ABB RobotStudio station: 20204 CCSU ROS EGM.rspag

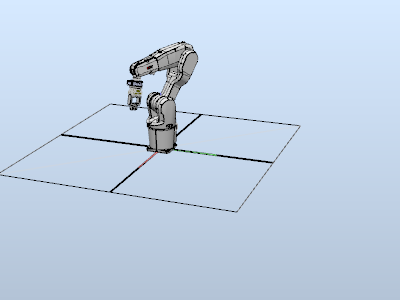
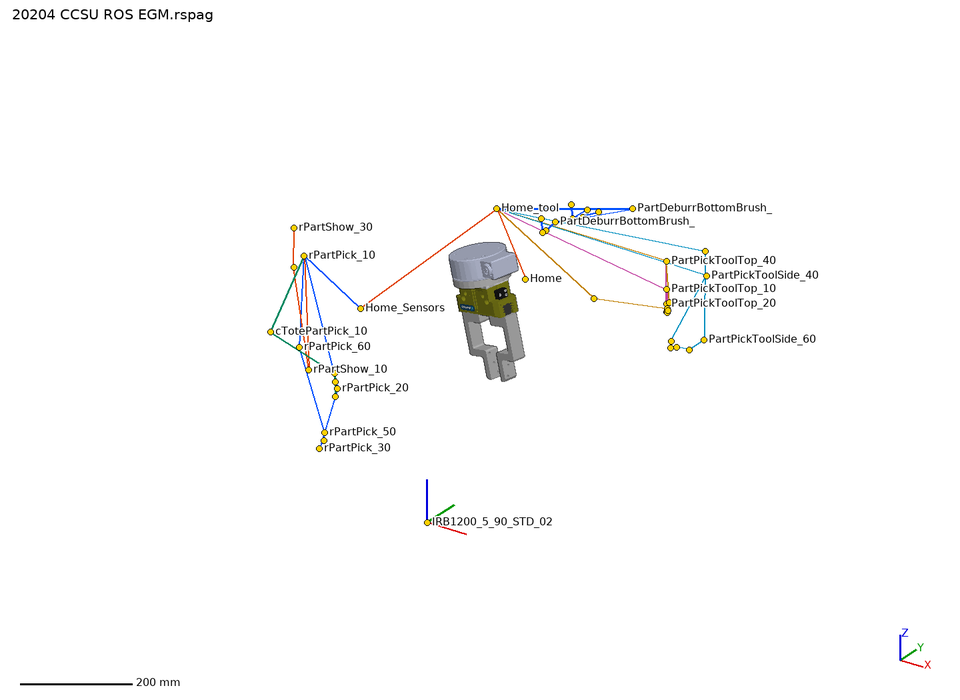
[picture v1: parts stored in the station drawn from their meshes, with robot base, taught points and paths (robot models come from the ABB library and are not in the file)]
--- station ---
Station 20204 CCSU RS (saved by RobotStudio 22.3.10098.0)
Controller 1200-800743_OfflineStation
  mechanical unit ROB_1: IRB1200_5_90_STD_02, 6 joints, base frame (0, 0, 0) mm
Layout (positions relative to the parent item):
  - IRB1200_5_90_STD_02 [mechanism, from %ABB.RobotStudio.Models.IRB1200%\IRB1200_5_90_STD_03.rslib] at (0, 0, 0) mm; joint values [-0.6243, -0.5477, 0.7485, -3.0114, -1.1483, -1.9775] (rad or m)
  - GRIPPER ONLY [part] at (196.51, -129.61, 653.41) mm, rotated rx -178.16 ry -14.43 rz -15 deg, size 125.6 x 50 x 198.4 mm
  - GRIPPER FORCE SENSOR [part] at (196.51, -129.61, 653.41) mm, rotated rx -178.16 ry -14.43 rz -15 deg, size 142.7 x 104 x 238.4 mm
Attachment: GRIPPER ONLY is attached to IRB1200_5_90_STD_02 / Link6
Attachment: GRIPPER FORCE SENSOR is attached to IRB1200_5_90_STD_02 / Link6
Targets, tools, work objects and paths stored in the station and not in the controller backup, written as RAPID:
! task T_ROB1
MODULE FORCENewProgram
  CONST robtarget GoHome:=[[-163.21,-220.75,679.83],[0.000017864,-0.460993,0.887404,0.000003505],[-2,0,1,0],[9E+09,9E+09,9E+09,9E+09,9E+09,9E+09]];
  PROC rGoHome()
    MoveJ GoHome,v500,z50,tool0;
  ENDPROC
ENDMODULE


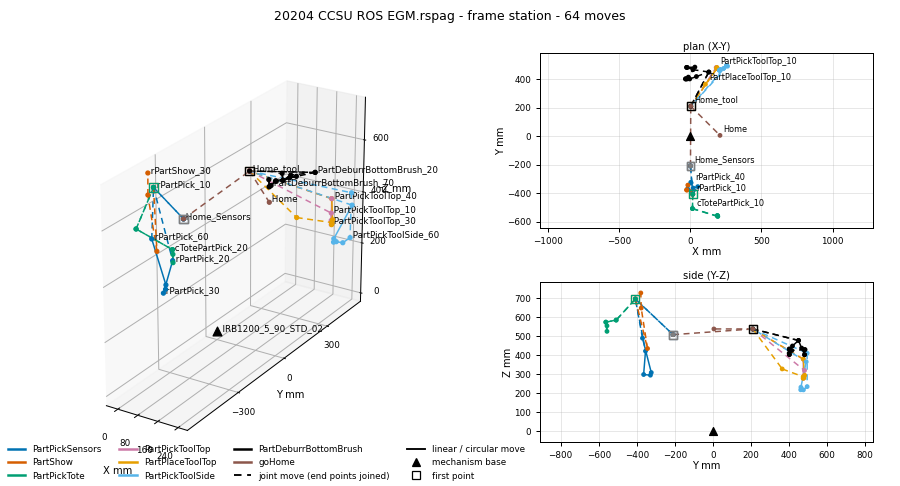
[picture p0: tool path of 20204 CCSU ROS EGM.rspag in frame station, 64 of 64 moves have a stored position in this frame; points joined in program order, loops and branches not executed]
--- Backups/1200-800743_OfflineStation/RAPID/TASK1/PROGMOD/CCSUMain.mod ---
MODULE CCSUMain
    CONST robtarget Home:=[[209.53,5.16,537.39],[0.00328327,0.0146564,-0.99987,0.00586276],[0,-1,-1,0],[9E+09,9E+09,9E+09,9E+09,9E+09,9E+09]];
    CONST robtarget Home_Sensors:=[[2.66,-209.51,507.39],[0.00651711,-0.708175,-0.706004,0.00177175],[-1,-1,0,0],[9E+09,9E+09,9E+09,9E+09,9E+09,9E+09]];
    CONST robtarget Home_tool:=[[4.44,209.54,537.36],[0.00162517,-0.701222,0.712912,-0.00653747],[0,-1,-1,0],[9E+09,9E+09,9E+09,9E+09,9E+09,9E+09]];

    CONST robtarget PartShowKeyence42_10:=[[6.27,-625.88,829.44],[0.494244,0.495626,0.505722,-0.504305],[-1,0,-1,1],[9E+09,9E+09,9E+09,9E+09,9E+09,9E+09]];

    CONST robtarget rPartPick_10:=[[18.54,-407.56,694.58],[0.00384471,-0.708054,0.706111,0.00724216],[-1,-1,2,0],[9E+09,9E+09,9E+09,9E+09,9E+09,9E+09]];
    CONST robtarget rPartPick_20:=[[53.83,-354.38,421.12],[0.499899,0.497617,-0.505452,0.496987],[-1,0,1,1],[9E+09,9E+09,9E+09,9E+09,9E+09,9E+09]];
    CONST robtarget rPartPick_30:=[[21.49,-364.23,297.89],[0.453944,0.556618,-0.376278,0.585258],[-2,-1,1,1],[9E+09,9E+09,9E+09,9E+09,9E+09,9E+09]];
    CONST robtarget rPartPick_40:=[[6.33,-328.65,294.34],[0.455745,0.555424,-0.377382,0.584281],[-2,-1,1,1],[9E+09,9E+09,9E+09,9E+09,9E+09,9E+09]];
    CONST robtarget rPartPick_50:=[[4.95,-324.08,308.23],[0.463269,0.542982,-0.36796,0.595951],[-2,-1,1,1],[9E+09,9E+09,9E+09,9E+09,9E+09,9E+09]];
    CONST robtarget rPartPick_60:=[[-17.82,-370.17,488.87],[0.449435,0.567565,-0.400681,0.561546],[-2,-1,2,1],[9E+09,9E+09,9E+09,9E+09,9E+09,9E+09]];

    CONST robtarget PartDeburrBottomBrush_10:=[[20.59,466.07,437.01],[0.602728,0.125692,-0.750355,-0.240599],[0,0,0,0],[9E+09,9E+09,9E+09,9E+09,9E+09,9E+09]];
    CONST robtarget PartDeburrBottomBrush_20:=[[131.20,449.67,476.97],[0.272617,0.273039,-0.90518,-0.178268],[0,0,0,0],[9E+09,9E+09,9E+09,9E+09,9E+09,9E+09]];
    CONST robtarget PartDeburrBottomBrush_30:=[[-21.43,481.63,402.00],[0.629363,0.053374,-0.75379,-0.181256],[0,0,0,0],[9E+09,9E+09,9E+09,9E+09,9E+09,9E+09]];
    CONST robtarget PartDeburrBottomBrush_40:=[[-25.46,482.17,428.74],[0.629308,0.0533195,-0.753849,-0.181216],[0,0,0,0],[9E+09,9E+09,9E+09,9E+09,9E+09,9E+09]];
    CONST robtarget PartDeburrBottomBrush_50:=[[33.47,484.19,428.74],[0.629353,0.0534079,-0.753787,-0.181294],[0,0,0,0],[9E+09,9E+09,9E+09,9E+09,9E+09,9E+09]];
    CONST robtarget PartDeburrBottomBrush_60:=[[-12.38,413.96,424.25],[0.492486,-0.605556,-0.452148,0.431649],[0,0,1,0],[9E+09,9E+09,9E+09,9E+09,9E+09,9E+09]];
    CONST robtarget PartDeburrBottomBrush_70:=[[-22.50,400.55,409.83],[0.178115,-0.733386,-0.0522476,0.653981],[0,0,2,0],[9E+09,9E+09,9E+09,9E+09,9E+09,9E+09]];
    CONST robtarget PartDeburrBottomBrush_80:=[[-30.75,401.69,403.02],[0.17569,-0.713364,-0.0583396,0.6759],[0,0,2,0],[9E+09,9E+09,9E+09,9E+09,9E+09,9E+09]];
    CONST robtarget PartDeburrBottomBrush_90:=[[-32.46,400.96,430.63],[0.175705,-0.7134,-0.0582814,0.675864],[0,0,2,0],[9E+09,9E+09,9E+09,9E+09,9E+09,9E+09]];
    CONST robtarget PartDeburrBottomBrush_100:=[[-2.75,400.95,432.33],[0.223478,-0.707408,-0.109083,0.661613],[0,0,1,0],[9E+09,9E+09,9E+09,9E+09,9E+09,9E+09]];
    CONST robtarget PartDeburrBottomBrush_110:=[[44.13,418.00,447.95],[0.552822,-0.233141,-0.776315,0.193307],[0,0,0,0],[9E+09,9E+09,9E+09,9E+09,9E+09,9E+09]];

    CONST robtarget PartPickToolTop_10:=[[182.71,481.27,319.22],[2.81422E-05,0.252387,-0.967626,5.44977E-05],[0,-1,0,0],[9E+09,9E+09,9E+09,9E+09,9E+09,9E+09]];
    CONST robtarget PartPickToolTop_20:=[[184.19,479.05,291.57],[2.52464E-05,0.275963,-0.961168,5.72893E-05],[0,-1,0,0],[9E+09,9E+09,9E+09,9E+09,9E+09,9E+09]];
    CONST robtarget PartPickToolTop_30:=[[186.90,474.91,277.87],[5.31134E-05,0.287484,-0.957786,8.70098E-05],[0,-1,0,0],[9E+09,9E+09,9E+09,9E+09,9E+09,9E+09]];
    CONST robtarget PartPickToolTop_40:=[[186.90,474.90,378.79],[7.99451E-05,0.287469,-0.95779,0.000131325],[0,-1,0,0],[9E+09,9E+09,9E+09,9E+09,9E+09,9E+09]];
    CONST robtarget PartPickToolTop_50:=[[95.27,363.91,463.37],[0.000545139,-0.492715,0.870185,-0.00319877],[0,-1,0,0],[9E+09,9E+09,9E+09,9E+09,9E+09,9E+09]];

    CONST robtarget PartPlaceToolTop_10:=[[107.24,363.98,327.23],[0.000830186,-0.460527,0.887641,-0.00281925],[0,-1,0,0],[9E+09,9E+09,9E+09,9E+09,9E+09,9E+09]];
    CONST robtarget PartPlaceToolTop_20:=[[188.59,474.22,286.25],[0.000721765,-0.280126,0.959959,-0.00283513],[0,-1,0,0],[9E+09,9E+09,9E+09,9E+09,9E+09,9E+09]];
    CONST robtarget PartPlaceToolTop_30:=[[188.60,474.24,277.87],[0.000713492,-0.281875,0.959447,-0.00283385],[0,-1,0,0],[9E+09,9E+09,9E+09,9E+09,9E+09,9E+09]];
    CONST robtarget PartPlaceToolTop_40:=[[188.09,478.25,280.22],[0.0006451,-0.281919,0.959433,-0.00292647],[0,-1,0,0],[9E+09,9E+09,9E+09,9E+09,9E+09,9E+09]];
    CONST robtarget PartPlaceToolTop_50:=[[188.08,481.96,293.90],[0.000649877,-0.281907,0.959437,-0.00291178],[0,-1,0,0],[9E+09,9E+09,9E+09,9E+09,9E+09,9E+09]];

    CONST robtarget PartPickToolSide_10:=[[256.14,495.20,409.71],[0.636266,-0.225868,0.723003,0.146344],[1,-2,1,0],[9E+09,9E+09,9E+09,9E+09,9E+09,9E+09]];
    CONST robtarget PartPickToolSide_20:=[[212.73,468.00,218.72],[0.636279,-0.225846,0.722991,0.146378],[1,-2,2,0],[9E+09,9E+09,9E+09,9E+09,9E+09,9E+09]];
    CONST robtarget PartPickToolSide_30:=[[205.28,461.34,217.68],[0.637331,-0.253883,0.717265,0.121997],[1,-2,1,0],[9E+09,9E+09,9E+09,9E+09,9E+09,9E+09]];
    CONST robtarget PartPickToolSide_40:=[[262.33,490.31,364.84],[0.63627,-0.225865,0.722995,0.146372],[0,-2,1,0],[9E+09,9E+09,9E+09,9E+09,9E+09,9E+09]];
    CONST robtarget PartPickToolSide_50:=[[180.42,458.49,569.25],[1.78132E-05,0.978994,0.20389,-8.85849E-06],[0,-1,-2,0],[9E+09,9E+09,9E+09,9E+09,9E+09,9E+09]];

    CONST robtarget rPartShow_10:=[[-16.06,-343.79,434.41],[0.511275,0.499772,0.487462,-0.501205],[-2,-1,0,1],[9E+09,9E+09,9E+09,9E+09,9E+09,9E+09]];
    CONST robtarget rPartShow_20:=[[-25.33,-376.99,647.3],[0.491571,0.508004,0.501758,-0.498527],[-2,-1,0,1],[9E+09,9E+09,9E+09,9E+09,9E+09,9E+09]];
    CONST robtarget rPartShow_30:=[[-22.55,-379.04,726.64],[0.57712,0.601052,0.394229,-0.387625],[-2,-1,0,1],[9E+09,9E+09,9E+09,9E+09,9E+09,9E+09]];

    CONST robtarget cTotePartPick_10:=[[16.46,-508.56,583.95],[0.0183208,-0.713973,0.699779,0.0147405],[-1,0,2,0],[9E+09,9E+09,9E+09,9E+09,9E+09,9E+09]];
    CONST robtarget cTotePartPick_20:=[[193.84,-562.84,573.2],[0.0180562,-0.70406,0.709754,0.0149481],[-1,0,2,0],[9E+09,9E+09,9E+09,9E+09,9E+09,9E+09]];
    CONST robtarget cTotePartPick_30:=[[191.27,-556.92,553.93],[0.0227291,-0.938112,0.345535,0.00595582],[-1,0,1,0],[9E+09,9E+09,9E+09,9E+09,9E+09,9E+09]];
    CONST robtarget cTotePartPick_40:=[[191.27,-556.92,524.77],[0.0227312,-0.938112,0.345535,0.00595572],[-1,0,1,0],[9E+09,9E+09,9E+09,9E+09,9E+09,9E+09]];
    CONST robtarget PartPickToolSide_60:=[[254.28,495.13,234.30],[0.636247,-0.225862,0.723024,0.146329],[1,-2,1,0],[9E+09,9E+09,9E+09,9E+09,9E+09,9E+09]];
    CONST robtarget PartPickToolSide_70:=[[235.72,475.43,217.08],[0.639167,-0.225261,0.720439,0.147279],[1,-2,2,0],[9E+09,9E+09,9E+09,9E+09,9E+09,9E+09]];
    CONST robtarget PartPickToolSide_80:=[[205.66,462.32,230.94],[0.639866,-0.244624,0.71687,0.129721],[1,-2,1,0],[9E+09,9E+09,9E+09,9E+09,9E+09,9E+09]];

    !TASK PERS tooldata CurrentTool:=[TRUE,[[0,0,228],[1,0,0,0]],[3.8,[-0.3,3.9,65.1],[1,0,0,0],0,0,0.006]]; !Totebox_GRIPPER_FS DATA !MOVED TO user SYSTEM MODULE



    !======================
    !=========MAIN=========
    !======================

    !PROC Main()
        !ForceStopRecording;
        !ForceLoadID;
        !ForceInitalization;
     !   MoveJ Home_Sensors,v100,fine,CurrentTool;


      !  VisionTest;
      !  goHome;
      !  PartDeburrBottomBrush;

       ! WaitTime 2;
       ! MoveJ Home_Sensors,v100,fine,CurrentTool;
        !ForceStopRecording;
       ! Stop\AllMoveTasks;
    !ENDPROC

    !======================
    !=======MAIN END=======
    !======================




    !for picking up part from single part stand on uppr platform
    PROC PartPickSensors()
        MoveJ Home_Sensors,v100,fine,CurrentTool;

        !part Home point
        MoveJ rPartPick_10,v500,z50,tool0;
        !move to Part
        MoveJ rPartPick_20,v500,fine,tool0;
        !move to pickup pre-orientation
        MoveL rPartPick_30,v100,fine,tool0;

        rGripperOpen;

        MoveL rPartPick_40,v40,fine,tool0;
        WaitTime 1.5;
        !grabing and correcting the part orientation
        rGripperClose;
        rGripperOpen;
        rGripperClose;
        WaitTime 1.5;

        MoveL rPartPick_50,v100,z50,tool0;
        MoveL rPartPick_60,v100,z50,tool0;
        MoveJ rPartPick_10,v500,z50,tool0;
        MoveJ Home_Sensors,v100,fine,CurrentTool;
    ENDPROC



    !for showing off grabbed items to the CognexCamera
    PROC PartShow()
        !part Home point
        MoveJ rPartPick_10,v500,z50,tool0;
        !show start position
        MoveJ rPartShow_10,v30,z50,tool0;
        MoveJ rPartShow_20,v30,z50,tool0;
        MoveJ rPartShow_30,v30,z50,tool0;
        !take photo_1



    ENDPROC


    !to pickup and place items from tote slot B8 (lower left corner) and returns to part pick Home
    PROC PartPickTote()
        !move to part pick Home
        MoveJ rPartPick_10,v100,z50,tool0;

        !get into position
        MoveJ cTotePartPick_10,v100,z50,tool0;
        !move to selection level
        MoveJ cTotePartPick_20,v100,z50,tool0;
        !move above slot B8
        rGripperOpen;

        !grab
        MoveL cTotePartPick_30,v30,z30,tool0;
        !orientate
        MoveL cTotePartPick_40,v10,z10,tool0;
        !move downward to pickup part
        rGripperClose;

        !return to part Home
        MoveL cTotePartPick_20,v100,z10,tool0;
        MoveJ cTotePartPick_10,v100,z50,tool0;
        MoveJ rPartPick_10,v100,z50,tool0;

    ENDPROC



    !picks up the bracket when placed on the tool plate and picking up from the top.
    PROC PartPickToolTop()

        MoveJ Home_tool,v500,z50,CurrentTool;

        MoveJ PartPickToolTop_10,v150,z50,CurrentTool;
        rGripperOpen;
        MoveL PartPickToolTop_20,v10,fine,CurrentTool;
        MoveL PartPickToolTop_30,v5,fine,CurrentTool;
        rGripperClose;
        WaitTime\InPos,1;
        MoveL PartPickToolTop_40,v150,z0,CurrentTool;

        MoveJ Home_tool,v500,z50,CurrentTool;


    ENDPROC



    !places a part back on the tool plate when gripping upright
    PROC PartPlaceToolTop()

        MoveJ Home_tool,v500,z50,CurrentTool;

        MoveJ PartPlaceToolTop_10,v150,z50,CurrentTool;
        MoveJ PartPlaceToolTop_20,v80,z50,CurrentTool;
        MoveJ PartPlaceToolTop_30,v5,z50,CurrentTool;
        WaitTime\InPos,1;
        rGripperOpen;
        MoveJ PartPlaceToolTop_40,v30,fine,CurrentTool;
        MoveJ PartPlaceToolTop_50,v30,fine,CurrentTool;

        MoveL PartPickToolTop_40,v150,z0,CurrentTool;


        MoveJ Home_tool,v500,z50,CurrentTool;


    ENDPROC



    !picks up the part on the tool plate from the side.
    PROC PartPickToolSide()

        MoveJ Home_tool,v500,z50,CurrentTool;

        MoveJ PartPickToolSide_10,v150,z50,CurrentTool;
        MoveJ PartPickToolSide_60,v40,z50,CurrentTool;
        MoveL PartPickToolSide_70,v20,z50,CurrentTool;
        rGripperOpen;
        MoveL PartPickToolSide_20,v10,fine,CurrentTool;
        MoveL PartPickToolSide_30,v5,fine,CurrentTool;
        WaitTime\InPos,1;
        rGripperClose;
        MoveL PartPickToolSide_80,v5,fine,CurrentTool;
        MoveL PartPickToolSide_40,v150,z0,CurrentTool;

        MoveJ Home_tool,v500,z50,CurrentTool;

    ENDPROC



    !deburrs the bottom edge of the part above the lettering with the brush
    PROC PartDeburrBottomBrush()

        !due to spindle speeds brush waits for all doors to be closed
        WaitDI DILeftDoorClosed,1;
        WaitDI DimiddleDoorClosed,1;
        WaitDI DIRightDoorClosed,1;

        rRunAtiTool;

        ! move close to tool.
        MoveJ Home_tool,v500,z50,CurrentTool;
        MoveJ PartDeburrBottomBrush_20,v150,z50,CurrentTool;
        MoveJ PartDeburrBottomBrush_10,v150,z50,CurrentTool;

        !slowly move from top down to deburr bottom side.
        MoveJ PartDeburrBottomBrush_30,v30,fine,CurrentTool;
        Movel PartDeburrBottomBrush_40,v5,fine,CurrentTool;
        MoveL PartDeburrBottomBrush_30,v5,fine,CurrentTool;

        !flip part deburr angle.
        MoveJ PartDeburrBottomBrush_50,v80,z50,CurrentTool;
        MoveJ PartDeburrBottomBrush_60,v150,z50,CurrentTool;
        MoveJ PartDeburrBottomBrush_70,v150,z50,CurrentTool;

        !Move from top down to deburr opposite side.
        MoveJ PartDeburrBottomBrush_80,v5,fine,CurrentTool;
        MoveL PartDeburrBottomBrush_90,v5,fine,CurrentTool;
        MoveL PartDeburrBottomBrush_80,v5,fine,CurrentTool;
        MoveJ PartDeburrBottomBrush_100,v50,z50,CurrentTool;


        !move away and back to Tool home
        MoveJ PartDeburrBottomBrush_110,v50,z50,CurrentTool;
        rStopRunAtiTool;
        MoveJ PartDeburrBottomBrush_20,v150,z50,CurrentTool;
        MoveJ Home_tool,v500,z50,CurrentTool;

    ENDPROC



    ! this program will show edge 42 of previously grabbed vane to the keyence sensor for instpection. IT RETURNS BACK TO HOME_SENSORS WHEN DONE.
    !PROC PartShowKeyence42()

    !    MoveJ Home_Sensors, v50, z50, CurrentTool;
    !    MoveJ PartShowKeyence42_10,v500,z50,CurrentTool;

    !    WaitRob\ZeroSpeed;
    !    KeyenceTrigger;
    !    WaitDI DI2KeyenceBusy,1;!TILL NOT BUSY FALLING EDGE AND WAIT HALF A SECOND
    !    WaitDI DI2KeyenceBusy,0;
    !    WaitTime(0.5);
    !
    !
    !    MoveJ Home_Sensors, v50, z50, CurrentTool;
    !
    !ENDPROC



ENDMODULE

--- Backups/1200-800743_OfflineStation/RAPID/TASK1/PROGMOD/Tooling.mod ---
MODULE Tooling
	CONST robtarget test123:=[[138.22,-7.70,799.49],[0.00599834,-0.565935,-0.332096,-0.754582],[-1,-1,-2,1],[9E+9,9E+9,9E+9,9E+9,9E+9,9E+9]];


    PROC rRunAtiTool()
        SetDO DOAtiSpindleCompSMC6,1;
        WaitTime\InPos,1;
        SetDO DOAtiSpindleStartSMC4,1;
    ENDPROC

    PROC rGripperClose()
        SetDO DOGripperCloseSMC0,0;
    ENDPROC

    PROC rGripperOpen()
        SetDO DOGripperCloseSMC0,1;
    ENDPROC

    FUNC bool rGripperIsOpen()
        IF(DOGripperCloseSMC0 = 1) THEN
            RETURN TRUE;
        ENDIF
        RETURN FALSE;
    ENDFUNC

    PROC rStopRunAtiTool()
        SetDO DOAtiSpindleStartSMC4,0;
        WaitTime 1;
        SetDO DOAtiSpindleCompSMC6,0;
    ENDPROC

    !PROC KeyenceTrigger()
    !    SetDO DO1KeyenceTrigger,1;
    !    WaitTime(0.01);
    !    SetDO DO1KeyenceTrigger,0;
    !ENDPROC

    PROC goHome()

        VAR pos CurrentPose;
        CurrentPose:=CPos(\Tool:=tool0\WObj:=wobj0);

        IF CurrentPose.y<-200 THEN
            MoveJ Home_Sensors,v500,z10,Gripper_FS;
        ENDIF

        IF CurrentPose.y>120 THEN
            MoveJ Home_Tool,v500,z10,Gripper_FS;
        ENDIF

        IF CurrentPose.x>0 THEN
            MoveJ Home,v500,z10,Gripper_FS;
        ENDIF

    ENDPROC

ENDMODULE

--- Backups/1200-800743_OfflineStation/RAPID/TASK1/PROGMOD/TRob1Main.mod ---
MODULE TRob1Main
    !***********************************************************
    ! Program data
    !***********************************************************
    ! Home position.
    LOCAL CONST jointtarget home := [[0, -30, 30, 0, 90, 0], [9E9, 9E9, 9E9, 9E9, 9E9, 9E9]];

    ! Identifier for the EGM correction.
    LOCAL VAR egmident egm_id;

    ! Limits for convergance.
    LOCAL VAR egm_minmax egm_condition := [-0.01, 0.01];

    ! EGM pose frames.
    LOCAL CONST pose egm_correction_frame := [[0, 0, 0], [1, 0, 0, 0]];
    LOCAL CONST pose egm_sensor_frame     := [[0, 0, 0], [1, 0, 0, 0]];

    ! The work object (here set to coincidence with ROB_2's base frame).
    LOCAL PERS wobjdata egm_wobj := [FALSE, TRUE, "", [[0, 1000, 0],[1, 0, 0, 0]], [[0, 0, 0],[1, 0, 0, 0]]];

    PROC main()
        TPWrite "Entered main()";
        MoveL Home_Sensors, v200, fine, tool0;

        ! Register an EGM id.
        EGMGetId egm_id;

        ! Setup the EGM communication.
        EGMSetupUC ROB_1, egm_id, "default", "ROB_1", \Pose;

        WHILE TRUE DO
            ! Prepare for an EGM communication session.
            EGMActPose egm_id,
                       \WObj:=wobj0,
                       egm_correction_frame,
                       EGM_FRAME_BASE,
                       egm_sensor_frame,
                       EGM_FRAME_BASE
                       \X:=egm_condition
                       \Y:=egm_condition
                       \Z:=egm_condition
                       \Rx:=egm_condition
                       \Ry:=egm_condition
                       \Rz:=egm_condition
                       \MaxSpeedDeviation:=100.0;

            ! Start the EGM communication session.
            ! EGMRunPose egm_id, EGM_STOP_RAMP_DOWN, \X \Y \Z \Rx \Ry \Rz \CondTime:=5 \RampOutTime:=5;

            !EGMRunPose egm_id, EGM_STOP_RAMP_DOWN, \X \Y \Z \CondTime:=30 \RampOutTime:=5;
            !TPWrite "Movising to position";
            EGMRunPose egm_id, EGM_STOP_HOLD, \X \Y \Z \Rx \Ry \Rz \CondTime:=0.01 \RampInTime:=0.05 \RampOutTime:=0.05;! \PosCorrGain:=0;

            !WaitTime 0.05;
        ENDWHILE

        ! Release the EGM id.
            EGMReset egm_id;
    ERROR
        IF ERRNO = ERR_UDPUC_COMM THEN
            TPWrite "Communication timedout";
            TRYNEXT;
        ENDIF
    ENDPROC

ENDMODULE

--- Backups/1200-800743_OfflineStation/RAPID/TASK1/SYSMOD/user.sys ---
MODULE user (SYSMODULE)

 ! Predefined user data
 !*********************

 ! Declaration of numeric registers reg1...reg5
 VAR num reg1 := 0;
 VAR num reg2 := 0;
 VAR num reg3 := 0;
 VAR num reg4 := 0;
 VAR num reg5 := 0;

 ! Declaration of stopwatch clock1
 VAR clock clock1;

  !TOOL DATA
    TASK PERS tooldata Gripper:=[TRUE,[[0,0,170],[1,0,0,0]],[1,[0,0,1],[1,0,0,0],0,0,0]];
    TASK PERS tooldata Gripper_FS:=[TRUE,[[0,0,225],[1,0,0,0]],[4,[-2.2,4.3,81.2],[1,0,0,0],0,0,0.006]];
    TASK PERS tooldata Gripper_Teach_FS:=[TRUE,[[0.248527,2.29601,199.301],[1,-0.000197831,7.9931E-05,2.1E-08]],[3.8,[5.6,5.4,66.9],[1,0,0,0],0,0.001,0.008]];
    TASK PERS tooldata Stationary_Spindle:=[FALSE,[[-175.829,466.985,420.318],[0.000147841,0.00108108,-0.000796757,0.999999]],[1,[0,0,0],[1,0,0,0],0,0,0]];
    TASK PERS tooldata Totebox_Gripper_FS:=[TRUE,[[0,0,228],[1,0,0,0]],[3.8,[-0.3,3.9,65.1],[1,0,0,0],0,0,0.006]];

    !WOBJ DATA
    TASK PERS wobjdata wobj4_partPlate:=[FALSE,TRUE,"",[[31.3314,-568.836,262.396],[1,2.39832E-05,-1.7637E-05,-0.000966885]],[[0,0,0],[1,0,0,0]]];
    TASK PERS wobjdata wobj3_highPlate:=[FALSE,TRUE,"",[[290.638,-318.993,133.1],[0.000175488,0.000151971,-0.000915474,-1]],[[0,0,0],[1,0,0,0]]];
    TASK PERS wobjdata wobj2_lowPlate:=[FALSE,TRUE,"",[[345.233,676.595,95.7232],[0.000865514,0.00117264,0.00221696,-0.999996]],[[0,0,0],[1,0,0,0]]];
    TASK PERS wobjdata wobj1_Spindle:=[FALSE,TRUE,"",[[-175.829,466.985,420.318],[8.88693E-05,-1,-0.000878471,7.79709E-05]],[[1.42852,-14.1366,-192.589],[0.00161154,0.706987,-0.707225,-9.07305E-05]]];
    TASK PERS wobjdata CamWobj:=[FALSE,TRUE,"",[[-21.766,-454.896,254.679],[1,0.000166484,-1.29905E-05,0.000133382]],[[-27.1315,-74.5063,0],[0.999988,0,0,-0.00488688]]];



    !==========================
    !====USER CONTROL DATA=====
    !==========================

    !DEFAULT MOVE SPEED DATA (CHANGE x SUCH THAT [x,500,5000,1000] )
    VAR speeddata defaultmovespeed := [60,500,5000,1000];

    !COPPY AND PASTE TOOL DATA TO HERE, MAKE SURE TO RENAME TOOL.
    TASK PERS tooldata CurrentTool:=[TRUE,[[0,0,0],[1,0,0,0]],[0.001,[0,0,0.001],[1,0,0,0],0,0,0]]; !Totebox_GRIPPER_FS DATA

ENDMODULE

--- Backups/1200-800743_OfflineStation/HOME/ROS/rapid/ROS_motion.mod ---
MODULE ROS_motion

! Software License Agreement (BSD License)
!
! Copyright (c) 2012, Edward Venator, Case Western Reserve University
! Copyright (c) 2012, Jeremy Zoss, Southwest Research Institute
! All rights reserved.
!
! Redistribution and use in source and binary forms, with or without modification,
! are permitted provided that the following conditions are met:
!
!   Redistributions of source code must retain the above copyright notice, this
!       list of conditions and the following disclaimer.
!   Redistributions in binary form must reproduce the above copyright notice, this
!       list of conditions and the following disclaimer in the documentation
!       and/or other materials provided with the distribution.
!   Neither the name of the Case Western Reserve University nor the names of its contributors
!       may be used to endorse or promote products derived from this software without
!       specific prior written permission.
!
! THIS SOFTWARE IS PROVIDED BY THE COPYRIGHT HOLDERS AND CONTRIBUTORS "AS IS" AND ANY
! EXPRESS OR IMPLIED WARRANTIES, INCLUDING, BUT NOT LIMITED TO, THE IMPLIED WARRANTIES
! OF MERCHANTABILITY AND FITNESS FOR A PARTICULAR PURPOSE ARE DISCLAIMED. IN NO EVENT
! SHALL THE COPYRIGHT HOLDER OR CONTRIBUTORS BE LIABLE FOR ANY DIRECT, INDIRECT,
! INCIDENTAL, SPECIAL, EXEMPLARY, OR CONSEQUENTIAL DAMAGES (INCLUDING, BUT NOT LIMITED
! TO, PROCUREMENT OF SUBSTITUTE GOODS OR SERVICES; LOSS OF USE, DATA, OR PROFITS; OR
! BUSINESS INTERRUPTION) HOWEVER CAUSED AND ON ANY THEORY OF LIABILITY, WHETHER IN
! CONTRACT, STRICT LIABILITY, OR TORT (INCLUDING NEGLIGENCE OR OTHERWISE) ARISING IN ANY
! WAY OUT OF THE USE OF THIS SOFTWARE, EVEN IF ADVISED OF THE POSSIBILITY OF SUCH DAMAGE.

LOCAL CONST zonedata DEFAULT_CORNER_DIST := z10;
LOCAL VAR ROS_joint_trajectory_pt trajectory{MAX_TRAJ_LENGTH};
LOCAL VAR num trajectory_size := 0;
LOCAL VAR intnum intr_new_trajectory;

PROC main()
    VAR num current_index;
    VAR jointtarget target;
    VAR speeddata move_speed := v10;  ! default speed
    VAR zonedata stop_mode;
    VAR bool skip_move;

    ! Set up interrupt to watch for new trajectory
    IDelete intr_new_trajectory;    ! clear interrupt handler, in case restarted with ExitCycle
    CONNECT intr_new_trajectory WITH new_trajectory_handler;
    IPers ROS_new_trajectory, intr_new_trajectory;

    WHILE true DO
        ! Check for new Trajectory
        IF (ROS_new_trajectory)
            init_trajectory;

        ! execute all points in this trajectory
        IF (trajectory_size > 0) THEN
            FOR current_index FROM 1 TO trajectory_size DO
                target.robax := trajectory{current_index}.joint_pos;
                target.extax := trajectory{current_index}.extax_pos;

                skip_move := (current_index = 1) AND is_near(target, 0.1, 0.1);

                stop_mode := DEFAULT_CORNER_DIST;  ! assume we're smoothing between points
                IF (current_index = trajectory_size) stop_mode := fine;  ! stop at path end

                ! Execute move command
                IF (NOT skip_move)
                    MoveAbsJ target, move_speed, \T:=trajectory{current_index}.duration, stop_mode, tool0;
            ENDFOR

            trajectory_size := 0;  ! trajectory done
        ENDIF

        WaitTime 0.05;  ! Throttle loop while waiting for new command
    ENDWHILE
ERROR
    ErrWrite \W, "Motion Error", "Error executing motion.  Aborting trajectory.";
    abort_trajectory;
ENDPROC

LOCAL PROC init_trajectory()
    clear_path;                    ! cancel any active motions

    WaitTestAndSet ROS_trajectory_lock;  ! acquire data-lock
    trajectory := ROS_trajectory;            ! copy to local var
    trajectory_size := ROS_trajectory_size;  ! copy to local var
    ROS_new_trajectory := FALSE;
    ROS_trajectory_lock := FALSE;         ! release data-lock
ENDPROC

LOCAL FUNC bool is_near(jointtarget target, num deg_tol, num mm_tol)
    VAR jointtarget curr_jnt;

    curr_jnt := CJointT();

    ! either an external axis is unconfigured/not present OR if it is, then it must be close enough
    RETURN ( ABS(curr_jnt.robax.rax_1 - target.robax.rax_1) < deg_tol )
       AND ( ABS(curr_jnt.robax.rax_2 - target.robax.rax_2) < deg_tol )
       AND ( ABS(curr_jnt.robax.rax_3 - target.robax.rax_3) < deg_tol )
       AND ( ABS(curr_jnt.robax.rax_4 - target.robax.rax_4) < deg_tol )
       AND ( ABS(curr_jnt.robax.rax_5 - target.robax.rax_5) < deg_tol )
       AND ( ABS(curr_jnt.robax.rax_6 - target.robax.rax_6) < deg_tol )
       AND ( (curr_jnt.extax.eax_a = 9E9) OR (ABS(curr_jnt.extax.eax_a - target.extax.eax_a) < mm_tol) )
       AND ( (curr_jnt.extax.eax_b = 9E9) OR (ABS(curr_jnt.extax.eax_b - target.extax.eax_b) < mm_tol) )
       AND ( (curr_jnt.extax.eax_c = 9E9) OR (ABS(curr_jnt.extax.eax_c - target.extax.eax_c) < mm_tol) )
       AND ( (curr_jnt.extax.eax_d = 9E9) OR (ABS(curr_jnt.extax.eax_d - target.extax.eax_d) < mm_tol) );
ENDFUNC

LOCAL PROC abort_trajectory()
    trajectory_size := 0;  ! "clear" local trajectory
    clear_path;
    ExitCycle;  ! restart program
ENDPROC

LOCAL PROC clear_path()
    IF ( NOT (IsStopMoveAct(\FromMoveTask) OR IsStopMoveAct(\FromNonMoveTask)) )
        StopMove;          ! stop any active motions
    ClearPath;             ! clear queued motion commands
    StartMove;             ! re-enable motions
ENDPROC

LOCAL TRAP new_trajectory_handler
    IF (NOT ROS_new_trajectory) RETURN;

    abort_trajectory;
ENDTRAP

ENDMODULE

--- Backups/1200-800743_OfflineStation/HOME/ROS/rapid/ROS_motionServer.mod ---
MODULE ROS_motionServer

! Software License Agreement (BSD License)
!
! Copyright (c) 2012, Edward Venator, Case Western Reserve University
! Copyright (c) 2012, Jeremy Zoss, Southwest Research Institute
! All rights reserved.
!
! Redistribution and use in source and binary forms, with or without modification,
! are permitted provided that the following conditions are met:
!
!   Redistributions of source code must retain the above copyright notice, this
!       list of conditions and the following disclaimer.
!   Redistributions in binary form must reproduce the above copyright notice, this
!       list of conditions and the following disclaimer in the documentation
!       and/or other materials provided with the distribution.
!   Neither the name of the Case Western Reserve University nor the names of its contributors
!       may be used to endorse or promote products derived from this software without
!       specific prior written permission.
!
! THIS SOFTWARE IS PROVIDED BY THE COPYRIGHT HOLDERS AND CONTRIBUTORS "AS IS" AND ANY
! EXPRESS OR IMPLIED WARRANTIES, INCLUDING, BUT NOT LIMITED TO, THE IMPLIED WARRANTIES
! OF MERCHANTABILITY AND FITNESS FOR A PARTICULAR PURPOSE ARE DISCLAIMED. IN NO EVENT
! SHALL THE COPYRIGHT HOLDER OR CONTRIBUTORS BE LIABLE FOR ANY DIRECT, INDIRECT,
! INCIDENTAL, SPECIAL, EXEMPLARY, OR CONSEQUENTIAL DAMAGES (INCLUDING, BUT NOT LIMITED
! TO, PROCUREMENT OF SUBSTITUTE GOODS OR SERVICES; LOSS OF USE, DATA, OR PROFITS; OR
! BUSINESS INTERRUPTION) HOWEVER CAUSED AND ON ANY THEORY OF LIABILITY, WHETHER IN
! CONTRACT, STRICT LIABILITY, OR TORT (INCLUDING NEGLIGENCE OR OTHERWISE) ARISING IN ANY
! WAY OUT OF THE USE OF THIS SOFTWARE, EVEN IF ADVISED OF THE POSSIBILITY OF SUCH DAMAGE.

LOCAL CONST num server_port := 11000;

LOCAL VAR socketdev server_socket;
LOCAL VAR socketdev client_socket;
LOCAL VAR ROS_joint_trajectory_pt trajectory{MAX_TRAJ_LENGTH};
LOCAL VAR num trajectory_size;

PROC main()
    VAR ROS_msg_joint_traj_pt message;

    TPWrite "MotionServer: Waiting for connection.";
    ROS_init_socket server_socket, server_port;
    ROS_wait_for_client server_socket, client_socket;

    WHILE ( true ) DO
        ! Recieve Joint Trajectory Pt Message
        ROS_receive_msg_joint_traj_pt client_socket, message;
        trajectory_pt_callback message;
    ENDWHILE

ERROR (ERR_SOCK_TIMEOUT, ERR_SOCK_CLOSED)
    IF (ERRNO=ERR_SOCK_TIMEOUT) OR (ERRNO=ERR_SOCK_CLOSED) THEN
        SkipWarn;  ! TBD: include this error data in the message logged below?
        ErrWrite \W, "ROS MotionServer disconnect", "Connection lost.  Resetting socket.";
        ExitCycle;  ! restart program
    ELSE
        TRYNEXT;
    ENDIF
UNDO
    IF (SocketGetStatus(client_socket) <> SOCKET_CLOSED) SocketClose client_socket;
    IF (SocketGetStatus(server_socket) <> SOCKET_CLOSED) SocketClose server_socket;
ENDPROC

LOCAL PROC trajectory_pt_callback(ROS_msg_joint_traj_pt message)
    VAR ROS_joint_trajectory_pt point;
    VAR jointtarget current_pos;
    VAR ROS_msg reply_msg;

    point := [message.joints, message.ext_axes, message.duration];

    ! use sequence_id to signal start/end of trajectory download
    TEST message.sequence_id
        CASE ROS_TRAJECTORY_START_DOWNLOAD:
            TPWrite "Traj START received";
            trajectory_size := 0;                 ! Reset trajectory size
            add_traj_pt point;                    ! Add this point to the trajectory
        CASE ROS_TRAJECTORY_END:
            TPWrite "Traj END received";
            add_traj_pt point;                    ! Add this point to the trajectory
            activate_trajectory;
        CASE ROS_TRAJECTORY_STOP:
            TPWrite "Traj STOP received";
            trajectory_size := 0;  ! empty trajectory
            activate_trajectory;
            StopMove; ClearPath; StartMove;  ! redundant, but re-issue stop command just to be safe
        DEFAULT:
            add_traj_pt point;                    ! Add this point to the trajectory
    ENDTEST

    ! send reply, if requested
    IF (message.header.comm_type = ROS_COM_TYPE_SRV_REQ) THEN
        reply_msg.header := [ROS_MSG_TYPE_JOINT_TRAJ_PT, ROS_COM_TYPE_SRV_REPLY, ROS_REPLY_TYPE_SUCCESS];
        ROS_send_msg client_socket, reply_msg;
    ENDIF

ERROR
    RAISE;  ! raise errors to calling code
ENDPROC

LOCAL PROC add_traj_pt(ROS_joint_trajectory_pt point)
    IF (trajectory_size = MAX_TRAJ_LENGTH) THEN
        ErrWrite \W, "Too Many Trajectory Points", "Trajectory has already reached its maximum size",
                 \RL2:="max_size = " + ValToStr(MAX_TRAJ_LENGTH);
    ELSE
        Incr trajectory_size;
        trajectory{trajectory_size} := point; !Add this point to the trajectory
    ENDIF
ENDPROC

LOCAL PROC activate_trajectory()
    WaitTestAndSet ROS_trajectory_lock;  ! acquire data-lock
    TPWrite "Sending " + ValToStr(trajectory_size) + " points to MOTION task";
    ROS_trajectory := trajectory;
    ROS_trajectory_size := trajectory_size;
    ROS_new_trajectory := TRUE;
    ROS_trajectory_lock := FALSE;  ! release data-lock
ENDPROC

ENDMODULE

--- Backups/1200-800743_OfflineStation/HOME/ROS/rapid/ROS_stateServer.mod ---
MODULE ROS_stateServer

! Software License Agreement (BSD License)
!
! Copyright (c) 2012, Edward Venator, Case Western Reserve University
! Copyright (c) 2012, Jeremy Zoss, Southwest Research Institute
! All rights reserved.
!
! Redistribution and use in source and binary forms, with or without modification,
! are permitted provided that the following conditions are met:
!
!   Redistributions of source code must retain the above copyright notice, this
!       list of conditions and the following disclaimer.
!   Redistributions in binary form must reproduce the above copyright notice, this
!       list of conditions and the following disclaimer in the documentation
!       and/or other materials provided with the distribution.
!   Neither the name of the Case Western Reserve University nor the names of its contributors
!       may be used to endorse or promote products derived from this software without
!       specific prior written permission.
!
! THIS SOFTWARE IS PROVIDED BY THE COPYRIGHT HOLDERS AND CONTRIBUTORS "AS IS" AND ANY
! EXPRESS OR IMPLIED WARRANTIES, INCLUDING, BUT NOT LIMITED TO, THE IMPLIED WARRANTIES
! OF MERCHANTABILITY AND FITNESS FOR A PARTICULAR PURPOSE ARE DISCLAIMED. IN NO EVENT
! SHALL THE COPYRIGHT HOLDER OR CONTRIBUTORS BE LIABLE FOR ANY DIRECT, INDIRECT,
! INCIDENTAL, SPECIAL, EXEMPLARY, OR CONSEQUENTIAL DAMAGES (INCLUDING, BUT NOT LIMITED
! TO, PROCUREMENT OF SUBSTITUTE GOODS OR SERVICES; LOSS OF USE, DATA, OR PROFITS; OR
! BUSINESS INTERRUPTION) HOWEVER CAUSED AND ON ANY THEORY OF LIABILITY, WHETHER IN
! CONTRACT, STRICT LIABILITY, OR TORT (INCLUDING NEGLIGENCE OR OTHERWISE) ARISING IN ANY
! WAY OUT OF THE USE OF THIS SOFTWARE, EVEN IF ADVISED OF THE POSSIBILITY OF SUCH DAMAGE.

LOCAL CONST num server_port := 11002;
LOCAL CONST num update_rate := 0.10;  ! broadcast rate (sec)

LOCAL VAR socketdev server_socket;
LOCAL VAR socketdev client_socket;

PROC main()

    TPWrite "StateServer: Waiting for connection.";
    ROS_init_socket server_socket, server_port;
    ROS_wait_for_client server_socket, client_socket;

    WHILE (TRUE) DO
        send_joints;
        send_status;
        WaitTime update_rate;
    ENDWHILE

ERROR (ERR_SOCK_TIMEOUT, ERR_SOCK_CLOSED)
    IF (ERRNO=ERR_SOCK_TIMEOUT) OR (ERRNO=ERR_SOCK_CLOSED) THEN
        SkipWarn;  ! TBD: include this error data in the message logged below?
        ErrWrite \W, "ROS StateServer disconnect", "Connection lost.  Waiting for new connection.";
        ExitCycle;  ! restart program
    ELSE
        TRYNEXT;
    ENDIF
UNDO
ENDPROC

LOCAL PROC send_joints()
    VAR ROS_msg_joint_data message;
    VAR jointtarget joints;

    ! get current joint position (degrees)
    joints := CJointT();

    ! create message
    message.header := [ROS_MSG_TYPE_JOINT, ROS_COM_TYPE_TOPIC, ROS_REPLY_TYPE_INVALID];
    message.sequence_id := 0;
    message.joints := joints.robax;
    message.ext_axes := joints.extax;

    ! send message to client
    ROS_send_msg_joint_data client_socket, message;

ERROR
    RAISE;  ! raise errors to calling code
ENDPROC

! signalExecutionError : System Output
! signalMotionPossible : System Output
! signalMotorOn : System Output
! signalRobotActive : System Output
! signalRobotEStop : System Output
! signalRobotNotMoving : System Output
! signalRosMotionTaskExecuting : System Output
LOCAL PROC send_status()
    VAR ROS_msg_robot_status message;

    ! get current joint position (degrees)
    ! joints := CJointT();

    ! create message
    message.header := [ROS_MSG_TYPE_STATUS, ROS_COM_TYPE_TOPIC, ROS_REPLY_TYPE_INVALID];
    message.sequence_id := 0;

    ! default values
    message.mode            := ROS_ROBOT_MODE_UNKNOWN;
    message.e_stopped       := ROS_TRISTATE_UNKNOWN;
    message.drives_powered  := ROS_TRISTATE_UNKNOWN;
    message.error_code      := ROS_TRISTATE_UNKNOWN;
    message.in_error        := ROS_TRISTATE_UNKNOWN;
    message.in_motion       := ROS_TRISTATE_UNKNOWN;
    message.motion_possible := ROS_TRISTATE_UNKNOWN;

    ! Get operating mode
    TEST OpMode()
        CASE OP_AUTO:
            message.mode := ROS_ROBOT_MODE_AUTO;
        CASE OP_MAN_PROG, OP_MAN_TEST:
            message.mode := ROS_ROBOT_MODE_MANUAL;
        CASE OP_UNDEF:
            message.mode := ROS_ROBOT_MODE_UNKNOWN;
    ENDTEST

    ! Get E-stop status
    IF DOutput(signalRobotEStop) = 1 THEN
        message.e_stopped := ROS_TRISTATE_ON;
    ELSE
        message.e_stopped := ROS_TRISTATE_OFF;
    ENDIF

    ! Get whether motors have power
    IF DOutput(signalMotorOn) = 1 THEN
        message.drives_powered := ROS_TRISTATE_TRUE;
    ELSE
        message.drives_powered := ROS_TRISTATE_FALSE;
    ENDIF

    ! Determine in_error and set error_code if in_error is true
    if DOutput(signalExecutionError) = 1 THEN
        message.in_error := ROS_TRISTATE_TRUE;
        message.error_code := ERRNO;
    ELSE
        message.in_error := ROS_TRISTATE_FALSE;
        message.error_code := 0;
    ENDIF

    ! Get in_motion
    IF DOutput(signalRobotNotMoving) = 1 THEN
        message.in_motion := ROS_TRISTATE_FALSE;
    ELSE
        message.in_motion := ROS_TRISTATE_TRUE;
    ENDIF

    ! Get whether motion is possible
    if (DOutput(signalMotionPossible) = 1) AND
       (DOutput(signalRobotActive) = 1) AND
       (DOutput(signalMotorOn) = 1) AND
       (DOutput(signalRosMotionTaskExecuting) = 1) THEN
        message.motion_possible := ROS_TRISTATE_TRUE;
    ELSE
        message.motion_possible := ROS_TRISTATE_FALSE;
    ENDIF

    ! send message to client
    ROS_send_msg_robot_status client_socket, message;

ERROR
    RAISE;  ! raise errors to calling code
ENDPROC

ENDMODULE

--- Backups/1200-800743_OfflineStation/SYSPAR/EIO.cfg ---
EIO:CFG_1.0:6:1::
#
SYSSIG_OUT:

      -Status "EmStop" -Signal "DOBuzzer"

      -Status "EmStop" -Signal "DORedLight"

      -Status "AutoOn" -Signal "DOGreenLight"
#
INDUSTRIAL_NETWORK:

      -Name "EtherNetIP" -Connection "Private Network"\
      -Label "EtherNet/IP Adapter Network"

      -Name "DeviceNet" -Label "DeviceNet Master/Slave Network" -Address "2"
#
EIO_CROSS:

      -Name "StackColorOrange" -Res "DOOrangeLight" -Act1 "DORedLight"\
      -Act1_invert  -Oper1 "AND" -Act2 "DOGreenLight" -Act2_invert

      -Name "LowAirPressure" -Res "DORedLight" -Act1 "DILowAirPressure"\
      -Act1_invert

      -Name "SafetyDoorLockAutoModeSwitch" -Res "DODoorLock" -Act1 "AUTO1"
#
ETHERNETIP_DEVICE:

      -Name "SMCAir20" -Address "192.168.1.20" -OutputAssembly 150\
      -InputAssembly 100 -ConfigurationAssembly 105 -OutputSize 4 -InputSize 2

      -Name "TurckBL20" -Address "192.168.125.40" -OutputAssembly 104\
      -InputAssembly 103 -ConfigurationAssembly 106 -OutputSize 16 -InputSize 16
#
DEVICENET_INTERNAL_DEVICE:

      -Name "DN_Internal_Device" -VendorName "ABB Robotics"\
      -ProductName "DeviceNet Internal Slave Device"
#
ETHERNETIP_INTERNAL_DEVICE:

      -Name "EN_Internal_Device" -VendorName "ABB Robotics"\
      -ProductName "EtherNet/IP Internal Adapter Device"
#
EIO_SIGNAL:

      -Name "DOGripperCloseSMC0" -SignalType "DO" -Device "SMCAir20"\
      -Label "SMCAir_0" -DeviceMap "0" -Access "All"

      -Name "SMC2OpenPort" -SignalType "DO" -Device "SMCAir20" -Label "SMCAir_2"\
      -DeviceMap "2" -Access "All"

      -Name "DOAtiSpindleStartSMC4" -SignalType "DO" -Device "SMCAir20"\
      -Label "SMCAir_4" -DeviceMap "4" -Access "All"

      -Name "DOAtiSpindleCompSMC6" -SignalType "DO" -Device "SMCAir20"\
      -Label "SMCAir_6" -DeviceMap "6" -Access "All"

      -Name "SMC8OpenPort" -SignalType "DO" -Device "SMCAir20" -Label "SMCAir_8"\
      -DeviceMap "8" -Access "All"

      -Name "DOBuzzer" -SignalType "DO" -Device "TurckBL20"\
      -Label "DOTurckBL20_1" -DeviceMap "16" -Access "All"

      -Name "DORedLight" -SignalType "DO" -Device "TurckBL20"\
      -Label "DOTurckBL20_2" -DeviceMap "17" -Access "All"

      -Name "DOOrangeLight" -SignalType "DO" -Device "TurckBL20"\
      -Label "DOTurckBL20_3" -DeviceMap "18" -Access "All"

      -Name "DOGreenLight" -SignalType "DO" -Device "TurckBL20"\
      -Label "DOTurckBL20_4" -DeviceMap "19" -Access "All"

      -Name "DODoorLock" -SignalType "DO" -Device "TurckBL20"\
      -Label "DOTurckBL20_5" -DeviceMap "20" -Access "All"

      -Name "DO6BL20" -SignalType "DO" -Device "TurckBL20"\
      -Label "DOTurckBL20_6" -DeviceMap "21"

      -Name "DO7BL20" -SignalType "DO" -Device "TurckBL20"\
      -Label "DOTurckBL20_7" -DeviceMap "22"

      -Name "DO8BL20" -SignalType "DO" -Device "TurckBL20"\
      -Label "DOTurckBL20_8" -DeviceMap "23"

      -Name "DO9BL20" -SignalType "DO" -Device "TurckBL20"\
      -Label "DOTurckBL20_9" -DeviceMap "24"

      -Name "DO10BL20" -SignalType "DO" -Device "TurckBL20"\
      -Label "DOTurckBL20_10" -DeviceMap "25"

      -Name "DO11BL20" -SignalType "DO" -Device "TurckBL20"\
      -Label "DOTurckBL20_11" -DeviceMap "26"

      -Name "DO12BL20" -SignalType "DO" -Device "TurckBL20"\
      -Label "DOTurckBL20_12" -DeviceMap "27"

      -Name "DO13BL20" -SignalType "DO" -Device "TurckBL20"\
      -Label "DOTurckBL20_13" -DeviceMap "28"

      -Name "DO14BL20" -SignalType "DO" -Device "TurckBL20"\
      -Label "DOTurckBL20_14" -DeviceMap "29"

      -Name "DO15BL20" -SignalType "DO" -Device "TurckBL20"\
      -Label "DOTurckBL20_15" -DeviceMap "30"

      -Name "DO16BL20" -SignalType "DO" -Device "TurckBL20"\
      -Label "DOTurckBL20_16" -DeviceMap "31"

      -Name "DILowAirPressure" -SignalType "DI" -Device "TurckBL20"\
      -Label "DITurckBL20_1" -DeviceMap "16"

      -Name "DI2BL20" -SignalType "DI" -Device "TurckBL20"\
      -Label "DITurckBL20_2" -DeviceMap "17"

      -Name "DIRightDoorClosed" -SignalType "DI" -Device "TurckBL20"\
      -Label "DITurckBL20_3" -DeviceMap "18"

      -Name "DIMiddleDoorClosed" -SignalType "DI" -Device "TurckBL20"\
      -Label "DITurckBL20_4" -DeviceMap "19"

      -Name "DILeftDoorClosed" -SignalType "DI" -Device "TurckBL20"\
      -Label "DITurckBL20_5" -DeviceMap "20"

      -Name "DI6BL20" -SignalType "DI" -Device "TurckBL20"\
      -Label "DITurckBL20_6" -DeviceMap "21"

      -Name "DI7BL20" -SignalType "DI" -Device "TurckBL20"\
      -Label "DITurckBL20_7" -DeviceMap "22"

      -Name "DI8BL20" -SignalType "DI" -Device "TurckBL20"\
      -Label "DITurckBL20_8" -DeviceMap "23"

      -Name "DI9BL20" -SignalType "DI" -Device "TurckBL20"\
      -Label "DITurckBL20_9" -DeviceMap "24"

      -Name "DI10BL20" -SignalType "DI" -Device "TurckBL20"\
      -Label "DITurckBL20_10" -DeviceMap "25"

      -Name "DI11BL20" -SignalType "DI" -Device "TurckBL20"\
      -Label "DITurckBL20_11" -DeviceMap "26"

      -Name "DI12BL20" -SignalType "DI" -Device "TurckBL20"\
      -Label "DITurckBL20_12" -DeviceMap "27"

      -Name "DI13BL20" -SignalType "DI" -Device "TurckBL20"\
      -Label "DITurckBL20_13" -DeviceMap "28"

      -Name "DI14BL20" -SignalType "DI" -Device "TurckBL20"\
      -Label "DITurckBL20_14" -DeviceMap "29"

      -Name "DI15BL20" -SignalType "DI" -Device "TurckBL20"\
      -Label "DITurckBL20_15" -DeviceMap "30"

      -Name "DI16BL20" -SignalType "DI" -Device "TurckBL20"\
      -Label "DITurckBL20_16" -DeviceMap "31"

      -Name "DO1ABB" -SignalType "DO" -Device "d652" -Label "DOAbb_1"\
      -DeviceMap "0"

      -Name "DI1ABB" -SignalType "DI" -Device "d652" -Label "D1ABB_1"\
      -DeviceMap "0"

      -Name "DI2ABB" -SignalType "DI" -Device "d652" -Label "D1ABB_2"\
      -DeviceMap "1"

      -Name "DI3ABB" -SignalType "DI" -Device "d652" -Label "D1ABB_3"\
      -DeviceMap "2"

      -Name "DI4ABB" -SignalType "DI" -Device "d652" -Label "D1ABB_4"\
      -DeviceMap "3"

      -Name "DI5ABB" -SignalType "DI" -Device "d652" -Label "D1ABB_5"\
      -DeviceMap "4"

      -Name "DO2ABB" -SignalType "DO" -Device "d652" -Label "DOAbb_2"\
      -DeviceMap "1"

      -Name "DO3ABB" -SignalType "DO" -Device "d652" -Label "DOAbb_3"\
      -DeviceMap "2"

      -Name "DO4ABB" -SignalType "DO" -Device "d652" -Label "DOAbb_4"\
      -DeviceMap "3"

      -Name "DO5ABB" -SignalType "DO" -Device "d652" -Label "DOAbb_5"\
      -DeviceMap "4"

      -Name "DO6ABB" -SignalType "DO" -Device "d652" -Label "DOAbb_6"\
      -DeviceMap "5"

      -Name "DO7ABB" -SignalType "DO" -Device "d652" -Label "DOAbb_7"\
      -DeviceMap "6"

      -Name "DO8ABB" -SignalType "DO" -Device "d652" -Label "DOAbb_8"\
      -DeviceMap "7"

      -Name "DO9ABB" -SignalType "DO" -Device "d652" -Label "DOAbb_9"\
      -DeviceMap "8"

      -Name "DO10ABB" -SignalType "DO" -Device "d652" -Label "DOAbb_10"\
      -DeviceMap "9"

      -Name "DO11ABB" -SignalType "DO" -Device "d652" -Label "DOAbb_11"\
      -DeviceMap "10"

      -Name "DO12ABB" -SignalType "DO" -Device "d652" -Label "DOAbb_12"\
      -DeviceMap "11"

      -Name "DO13ABB" -SignalType "DO" -Device "d652" -Label "DOAbb_13"\
      -DeviceMap "12"

      -Name "DO14ABB" -SignalType "DO" -Device "d652" -Label "DOAbb_14"\
      -DeviceMap "13"

      -Name "DO15ABB" -SignalType "DO" -Device "d652" -Label "DOAbb_15"\
      -DeviceMap "14"

      -Name "DO16ABB" -SignalType "DO" -Device "d652" -Label "DOAbb_16"\
      -DeviceMap "15"

      -Name "DI6ABB" -SignalType "DI" -Device "d652" -Label "D1ABB_6"\
      -DeviceMap "5"

      -Name "DI7ABB" -SignalType "DI" -Device "d652" -Label "D1ABB_7"\
      -DeviceMap "6"

      -Name "DI8ABB" -SignalType "DI" -Device "d652" -Label "D1ABB_8"\
      -DeviceMap "7"

      -Name "DI9ABB" -SignalType "DI" -Device "d652" -Label "D1ABB_9"\
      -DeviceMap "8"

      -Name "DI10ABB" -SignalType "DI" -Device "d652" -Label "D1ABB_10"\
      -DeviceMap "9"

      -Name "DI11ABB" -SignalType "DI" -Device "d652" -Label "D1ABB_11"\
      -DeviceMap "10"

      -Name "DI12ABB" -SignalType "DI" -Device "d652" -Label "D1ABB_12"\
      -DeviceMap "11"

      -Name "DI13ABB" -SignalType "DI" -Device "d652" -Label "D1ABB_13"\
      -DeviceMap "12"

      -Name "DI14ABB" -SignalType "DI" -Device "d652" -Label "D1ABB_14"\
      -DeviceMap "13"

      -Name "DI15ABB" -SignalType "DI" -Device "d652" -Label "D1ABB_15"\
      -DeviceMap "14"

      -Name "DI16ABB" -SignalType "DI" -Device "d652" -Label "D1ABB_16"\
      -DeviceMap "15"

      -Name "DIDoorLock" -SignalType "DI" -Access "All" -Invert
